// Swaps values of two variables
FUNCTION SwapByPointer
VAR_INPUT
	a : POINTER TO BYTE;
	b : POINTER TO BYTE;
	length : DINT;
END_VAR
VAR
	temp : POINTER TO BYTE;
END_VAR

temp := __NEW(BYTE, TO_UDINT(length));

MEMCPY(temp, a, TO_UDINT(length));
MEMCPY(a, b, TO_UDINT(length));
MEMCPY(b, temp, TO_UDINT(length));

__DELETE(temp);

END_FUNCTION

(* stored: Version 1.1.0.1
   POU SwapByPointer: Id {b35f0ba5-480b-005d-053a-a6bc01854ed8}, SpecialFunc None *)
